FUNCTION_BLOCK WarpAffine (* openCV warp affine *)
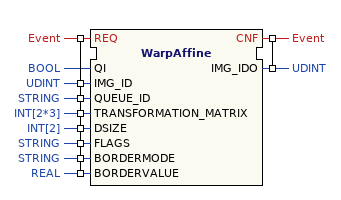
  EVENT_INPUT
    REQ WITH IMG_ID, QUEUE_ID, TRANSFORMATION_MATRIX, DSIZE, FLAGS, BORDERMODE, BORDERVALUE;
  END_EVENT
  EVENT_OUTPUT
    CNF WITH IMG_IDO;
  END_EVENT
  VAR_INPUT
    QI : BOOL;
    IMG_ID : UDINT;
    QUEUE_ID : STRING;
    TRANSFORMATION_MATRIX : ARRAY [2*3] OF INT;
    DSIZE : ARRAY [0..1] OF INT;
    FLAGS : STRING;
    BORDERMODE : STRING;
    BORDERVALUE : REAL;
  END_VAR
  VAR_OUTPUT
    IMG_IDO : UDINT;
  END_VAR
END_FUNCTION_BLOCK
